PROGRAM PRG_TEST
VAR
END_VAR

TcUnit.RUN();

END_PROGRAM

(* stored: Version 1.1.0.1, ProductVersion 3.1.4024.14
   POU PRG_TEST: Id {cb21ee53-cae2-46b9-9929-c0b774c55f6a}, SpecialFunc None *)
